// TwinCAT 3 PLC project MainPLC
// Title: IrrigationSystem
// Company: CleanGreens Solutions SA
// ProjectVersion: 0.5beat1
// ProgramVersion: 3.1.4024.0
// libraries:
//   Tc2_Database, * (Beckhoff Automation GmbH)
//   Tc2_DataExchange, * (Beckhoff Automation GmbH)
//   Tc2_IoFunctions, * (Beckhoff Automation GmbH)
//   Tc2_Math, * (Beckhoff Automation GmbH)
//   Tc2_MC2, * (Beckhoff Automation GmbH)
//   Tc2_Standard, * (Beckhoff Automation GmbH)
//   Tc2_SUPS, * (Beckhoff Automation GmbH)
//   Tc2_System, * (Beckhoff Automation GmbH)
//   Tc2_TcpIp, * (Beckhoff Automation GmbH)
//   Tc2_Utilities, * (Beckhoff Automation GmbH)
//   Tc2_XmlDataSrv, * (Beckhoff Automation GmbH)
//   Tc3_Database, * (Beckhoff Automation GmbH)
//   Tc3_EventLogger, * (Beckhoff Automation GmbH)
//   Tc3_Module, * (Beckhoff Automation GmbH)
// project tree:
//   DUTs/ ST_Robot_Axes.TcDUT (not stored)
//   GVLs/ C.TcGVL (not stored), G.TcGVL
//   / PlcTask.TcTTO (not stored)
//   POUs/ FB_PowerAxis1.TcPOU (not stored), FB_PowerMaster.TcPOU (not stored), Main.TcPOU
// real-time tasks:
//   TASK PlcTask: cycle T#10ms, priority 20, ADS port 350
//   TASK VISU_TASK: cycle T#200000us, priority 30, ADS port 351
// motion (NC):
//   TASK NC-Task 1 SAF: cycle T#2ms, priority 4, ADS port 501
//   TASK NC-Task 1 SVB: cycle T#10ms, priority 8, ADS port 511
//   AXIS CGSMini_Robot01AxisLine1Back (id 6)
//     General: UnitName=m
//     Dynamic: AccelerationMaximum=0.5, DecelerationMaximum=1.5, Acceleration=0.3, Deceleration=1, Jerk=0.33
//     Velo: RefSearch=0.01752, RefSync=0.01752, SlowManual=0.0876, FastManual=0.5256, Fast=1.752, Maximum=0.67
//     OtherSettings: AllowMotionCmdToSlave=true
//     encoder EncType=19
//       EncPara: ScaleFactorNumerator=0.79, ScaleFactorDenominator=26214400, Inverse=true, MaxCount=#xffffffff
//         ActPosCorrection: Enable=true, Time=1
//     drive DrvType=16
//       DrvPara: Inverse=true, MaxCount=#xffffffff, DriveControlDWord=#x00020100
//         Analog: VeloReferenz=0.737, VeloScale=71.5255737304688, TorqueSetpointScale=10, ScaleFactorActTorque=0.1
//         TimeComp: TaskDelayCycles=1
//     controller CtrType=1
//       CtrPara: PriorControlFactor=1
//         PosDiffControl: Range=0.1
//         Observer: BandWidth=20
//   AXIS CGSMini_Robot01AxisLine2Front (id 7)
//     General: UnitName=m
//     Dynamic: AccelerationMaximum=0.5, DecelerationMaximum=1.5, Acceleration=0.3, Deceleration=1, Jerk=0.33
//     Velo: RefSearch=0.01752, RefSync=0.01752, SlowManual=0.0876, FastManual=0.5256, Fast=1.752, Maximum=0.67
//     OtherSettings: AllowMotionCmdToSlave=true
//     encoder EncType=19
//       EncPara: ScaleFactorNumerator=0.79, ScaleFactorDenominator=26214400, Inverse=true, MaxCount=#xffffffff
//         ActPosCorrection: Enable=true, Time=1
//     drive DrvType=16
//       DrvPara: Inverse=true, MaxCount=#xffffffff, DriveControlDWord=#x00020100
//         Analog: VeloReferenz=0.737, VeloScale=71.5255737304688, TorqueSetpointScale=10, ScaleFactorActTorque=0.1
//         TimeComp: TaskDelayCycles=1
//     controller CtrType=1
//       CtrPara: PriorControlFactor=1
//         PosDiffControl: Range=0.1
//         Observer: BandWidth=20
//   AXIS CGSMini_Robot01AxisLine2Back (id 8)
//     General: UnitName=m
//     Dynamic: AccelerationMaximum=0.5, DecelerationMaximum=1.5, Acceleration=0.3, Deceleration=1, Jerk=0.33
//     Velo: RefSearch=0.01752, RefSync=0.01752, SlowManual=0.0876, FastManual=0.5256, Fast=1.752, Maximum=0.67
//     OtherSettings: AllowMotionCmdToSlave=true
//     encoder EncType=19
//       EncPara: ScaleFactorNumerator=0.79, ScaleFactorDenominator=26214400, Inverse=true, MaxCount=#xffffffff
//         ActPosCorrection: Enable=true, Time=1
//     drive DrvType=16
//       DrvPara: Inverse=true, MaxCount=#xffffffff, DriveControlDWord=#x00020100
//         Analog: VeloReferenz=0.737, VeloScale=71.5255737304688, TorqueSetpointScale=10, ScaleFactorActTorque=0.1
//         TimeComp: TaskDelayCycles=1
//     controller CtrType=1
//       CtrPara: PriorControlFactor=1
//         PosDiffControl: Range=0.1
//         Observer: BandWidth=20
//   AXIS CGSMini_Robot01AxisLine1Front (id 5)
//     General: UnitName=m
//     Dynamic: AccelerationMaximum=0.5, DecelerationMaximum=1.5, Acceleration=0.3, Deceleration=1, Jerk=0.33
//     Velo: RefSearch=0.01752, RefSync=0.01752, SlowManual=0.0876, FastManual=0.5256, Fast=1.752, Maximum=0.67
//     OtherSettings: AllowMotionCmdToSlave=true
//     encoder EncType=19
//       EncPara: ScaleFactorNumerator=0.79, ScaleFactorDenominator=26214400, Inverse=true, MaxCount=#xffffffff
//         ActPosCorrection: Enable=true, Time=1
//     drive DrvType=16
//       DrvPara: Inverse=true, MaxCount=#xffffffff, DriveControlDWord=#x00020100
//         Analog: VeloReferenz=0.737, VeloScale=71.5255737304688, TorqueSetpointScale=10, ScaleFactorActTorque=0.1
//         TimeComp: TaskDelayCycles=1
//     controller CtrType=1
//       CtrPara: PriorControlFactor=1
//         PosDiffControl: Range=0.1
//         Observer: BandWidth=20
//   AXIS CGSMini_Robot01AxisMaster (id 14)
//   AXIS Sim_Robot01AxisLine1Back (id 9)
//   AXIS Sim_Robot01AxisLine2Back (id 10)
//   AXIS Sim_Robot01AxisLine1Front (id 11)
//   AXIS Sim_Robot01AxisLine2Front (id 12)
//   AXIS Sim_Robot01AxisMaster (id 13)
// variable links:
//   MainPLC/MainPLC Instance <-> NC-Task 1 SAF/Axes/CGSMini_Robot01AxisLine1Back
//     PlcTask Inputs/G.stAX.Line1Back.NcToPlc <-> Outputs/ToPlc
//     PlcTask Outputs/G.stAX.Line1Back.PlcToNc <-> Inputs/FromPlc
//   MainPLC/MainPLC Instance <-> NC-Task 1 SAF/Axes/CGSMini_Robot01AxisLine1Front
//     PlcTask Inputs/G.stAX.Line1Front.NcToPlc <-> Outputs/ToPlc
//     PlcTask Outputs/G.stAX.Line1Front.PlcToNc <-> Inputs/FromPlc
//   MainPLC/MainPLC Instance <-> NC-Task 1 SAF/Axes/CGSMini_Robot01AxisLine2Back
//     PlcTask Inputs/G.stAX.Line2Back.NcToPlc <-> Outputs/ToPlc
//     PlcTask Outputs/G.stAX.Line2Back.PlcToNc <-> Inputs/FromPlc
//   MainPLC/MainPLC Instance <-> NC-Task 1 SAF/Axes/CGSMini_Robot01AxisLine2Front
//     PlcTask Inputs/G.stAX.Line2Front.NcToPlc <-> Outputs/ToPlc
//     PlcTask Outputs/G.stAX.Line2Front.PlcToNc <-> Inputs/FromPlc
//   MainPLC/MainPLC Instance <-> NC-Task 1 SAF/Axes/CGSMini_Robot01AxisMaster
//     PlcTask Inputs/G.stAX.Master.NcToPlc <-> Outputs/ToPlc
//     PlcTask Outputs/G.stAX.Master.PlcToNc <-> Inputs/FromPlc

// ---- GVLs/G.TcGVL
{attribute 'qualified_only'}
VAR_GLOBAL
  {attribute 'TcNcAxis' := '.Line1Front                       := CGSMini_Robot01AxisLine1Front;
                          .Line1Back                        := CGSMini_Robot01AxisLine1Back;
                          .Line2Front                       := CGSMini_Robot01AxisLine2Front;
                          .Line2Back                        := CGSMini_Robot01AxisLine2Back;
                          .Master                           := CGSMini_Robot01AxisMaster'}
  stAX : ST_Robot_Axes;
END_VAR

// ---- POUs/Main.TcPOU
PROGRAM Main
VAR
 	fbPowerMaster : FB_PowerMaster;
  fbPowerAxis1 : FB_PowerAxis1;
END_VAR

fbPowerMaster();

END_PROGRAM
